TYPE ST_System_MVHW_Zustand :
STRUCT
	Betrieb_Anford			: BOOL;
	Betrieb_Soll				: BOOL;
	Betrieb					: BOOL;

	Netze_Anford				: ST_Zustand_Netze_Anford;
	Netz_vorheizen			: BOOL;

	Freigabe					: BOOL;
	Freigabe_Deakt			: BOOL;
	Freigabe_Code			: WORD;

	Stoerung					: BOOL;
	Stoerung_Code			: WORD;

	Warnung					: BOOL;
	Warnung_Code			: WORD;

	Status					: SINT;
	Status_Vorl_Stellventil		: BOOL;
	Status_Vorl_Pumpe		: BOOL;
	Status_Nachl_Stellventil	: BOOL;
	Status_Nachl_Pumpe		: BOOL;

	Quittierung				: BOOL;

	Netz_HW_Anford			: ST_Zustand_Netz_Anford ; (* Philipp *)

END_STRUCT
END_TYPE

(* stored: Version 1.1.0.1, ProductVersion 3.1.4024.9
   DUT ST_System_MVHW_Zustand: Id {8b92e432-effe-4afc-986c-778e766d6d25} *)
